// TIA Portal V19 export
TYPE "TokenChain_Data"
// stored: Access Published
   STRUCT
      TOKEN : Int;
      USER : Int;
      OldToken : Int;
      TimeOut : IEC_TIMER;
   END_STRUCT;
END_TYPE
